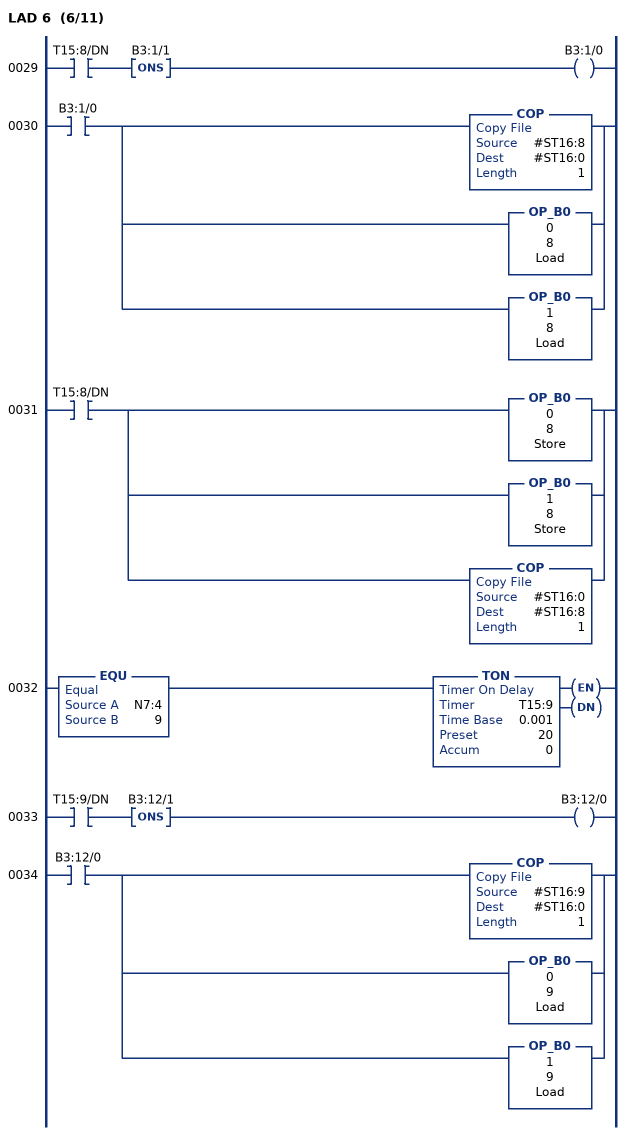
% Rung: 29 %
SOR XIC T15:8/DN ONS B3:1/1 OTE B3:1/0 EOR
% Rung: 30 %
SOR XIC B3:1/0 BST COP #ST16:8 #ST16:0 1 NXB OP_B0 0 8 Load NXB OP_B0 1 8 Load BND EOR
% Rung: 31 %
SOR XIC T15:8/DN BST OP_B0 0 8 Store NXB OP_B0 1 8 Store NXB COP #ST16:0 #ST16:8 1 BND EOR
% Rung: 32 %
SOR EQU N7:4 9 TON T15:9 0.001 20 0 EOR
% Rung: 33 %
SOR XIC T15:9/DN ONS B3:12/1 OTE B3:12/0 EOR
% Rung: 34 %
SOR XIC B3:12/0 BST COP #ST16:9 #ST16:0 1 NXB OP_B0 0 9 Load NXB OP_B0 1 9 Load BND EOR

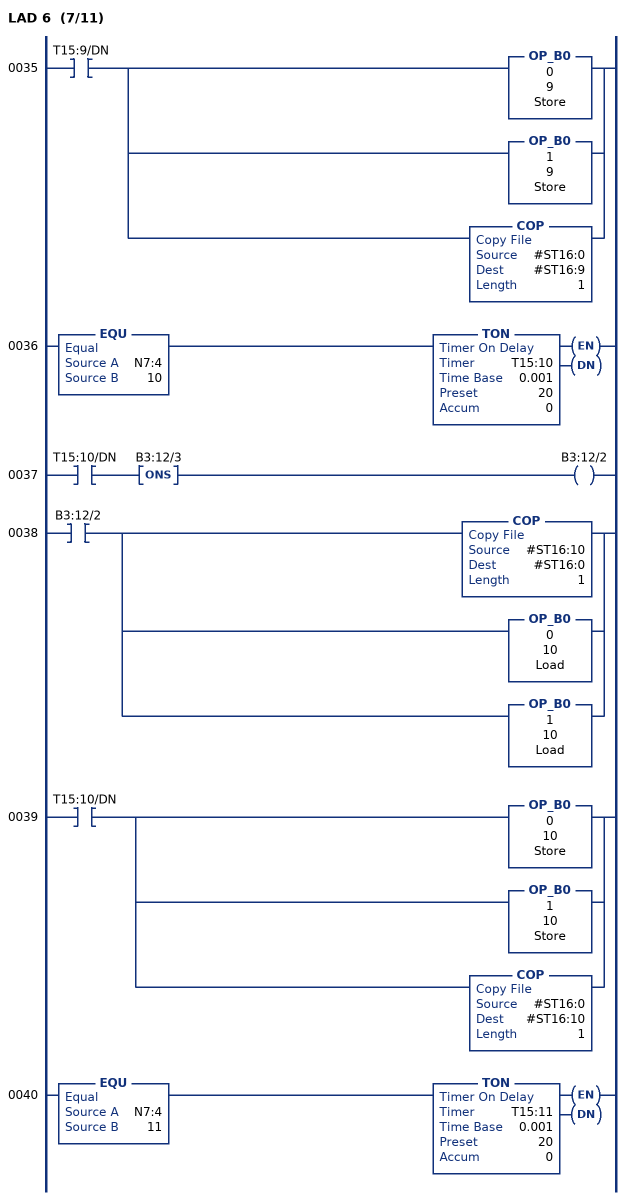
% Rung: 35 %
SOR XIC T15:9/DN BST OP_B0 0 9 Store NXB OP_B0 1 9 Store NXB COP #ST16:0 #ST16:9 1 BND EOR
% Rung: 36 %
SOR EQU N7:4 10 TON T15:10 0.001 20 0 EOR
% Rung: 37 %
SOR XIC T15:10/DN ONS B3:12/3 OTE B3:12/2 EOR
% Rung: 38 %
SOR XIC B3:12/2 BST COP #ST16:10 #ST16:0 1 NXB OP_B0 0 10 Load NXB OP_B0 1 10 Load BND EOR
% Rung: 39 %
SOR XIC T15:10/DN BST OP_B0 0 10 Store NXB OP_B0 1 10 Store NXB COP #ST16:0 #ST16:10 1 BND EOR
% Rung: 40 %
SOR EQU N7:4 11 TON T15:11 0.001 20 0 EOR

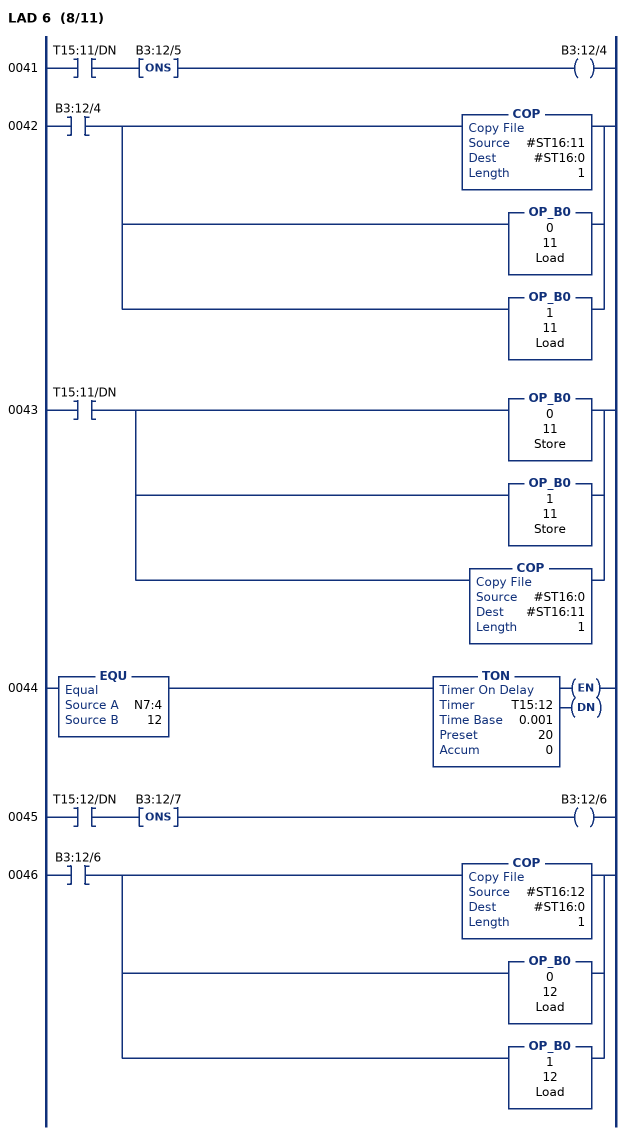
% Rung: 41 %
SOR XIC T15:11/DN ONS B3:12/5 OTE B3:12/4 EOR
% Rung: 42 %
SOR XIC B3:12/4 BST COP #ST16:11 #ST16:0 1 NXB OP_B0 0 11 Load NXB OP_B0 1 11 Load BND EOR
% Rung: 43 %
SOR XIC T15:11/DN BST OP_B0 0 11 Store NXB OP_B0 1 11 Store NXB COP #ST16:0 #ST16:11 1 BND EOR
% Rung: 44 %
SOR EQU N7:4 12 TON T15:12 0.001 20 0 EOR
% Rung: 45 %
SOR XIC T15:12/DN ONS B3:12/7 OTE B3:12/6 EOR
% Rung: 46 %
SOR XIC B3:12/6 BST COP #ST16:12 #ST16:0 1 NXB OP_B0 0 12 Load NXB OP_B0 1 12 Load BND EOR

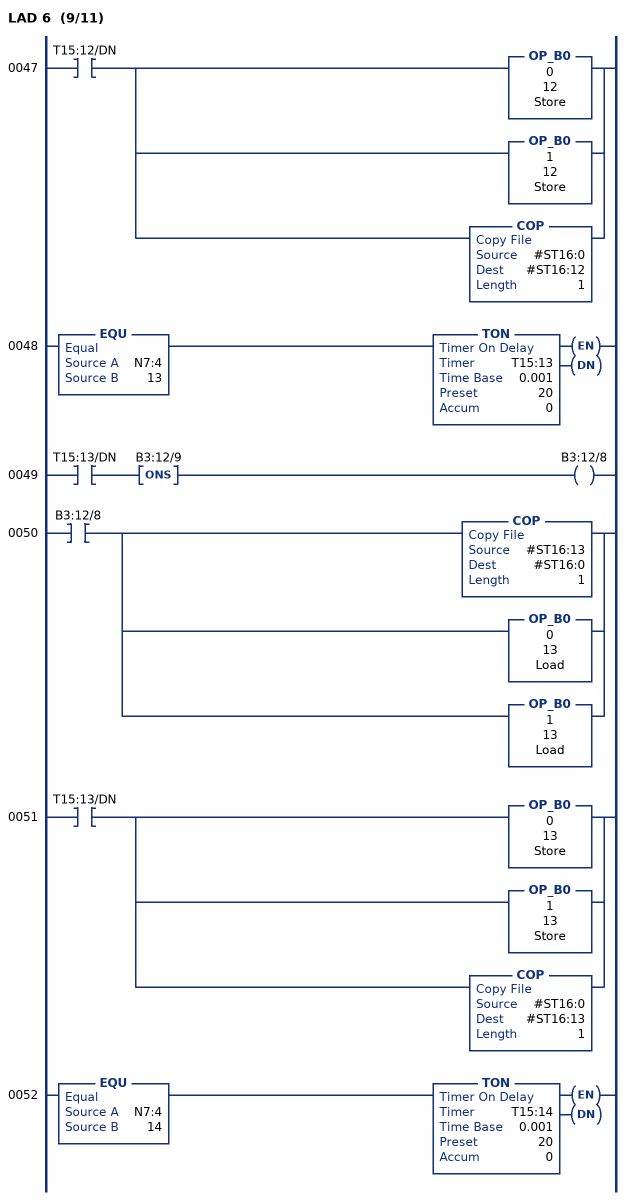
% Rung: 47 %
SOR XIC T15:12/DN BST OP_B0 0 12 Store NXB OP_B0 1 12 Store NXB COP #ST16:0 #ST16:12 1 BND EOR
% Rung: 48 %
SOR EQU N7:4 13 TON T15:13 0.001 20 0 EOR
% Rung: 49 %
SOR XIC T15:13/DN ONS B3:12/9 OTE B3:12/8 EOR
% Rung: 50 %
SOR XIC B3:12/8 BST COP #ST16:13 #ST16:0 1 NXB OP_B0 0 13 Load NXB OP_B0 1 13 Load BND EOR
% Rung: 51 %
SOR XIC T15:13/DN BST OP_B0 0 13 Store NXB OP_B0 1 13 Store NXB COP #ST16:0 #ST16:13 1 BND EOR
% Rung: 52 %
SOR EQU N7:4 14 TON T15:14 0.001 20 0 EOR

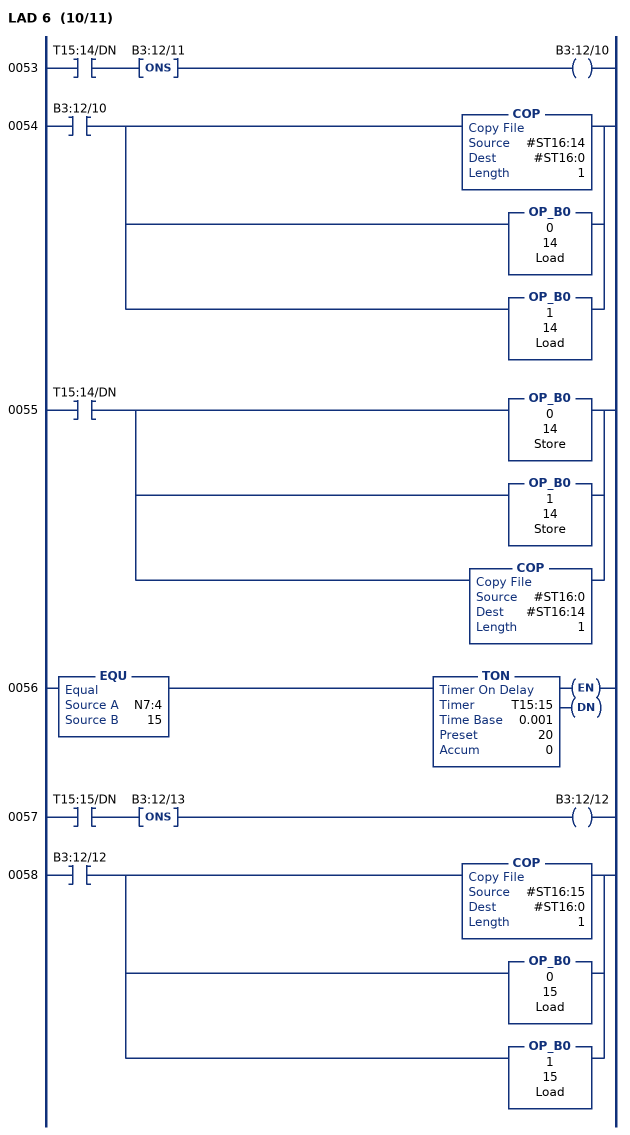
% Rung: 53 %
SOR XIC T15:14/DN ONS B3:12/11 OTE B3:12/10 EOR
% Rung: 54 %
SOR XIC B3:12/10 BST COP #ST16:14 #ST16:0 1 NXB OP_B0 0 14 Load NXB OP_B0 1 14 Load BND EOR
% Rung: 55 %
SOR XIC T15:14/DN BST OP_B0 0 14 Store NXB OP_B0 1 14 Store NXB COP #ST16:0 #ST16:14 1 BND EOR
% Rung: 56 %
SOR EQU N7:4 15 TON T15:15 0.001 20 0 EOR
% Rung: 57 %
SOR XIC T15:15/DN ONS B3:12/13 OTE B3:12/12 EOR
% Rung: 58 %
SOR XIC B3:12/12 BST COP #ST16:15 #ST16:0 1 NXB OP_B0 0 15 Load NXB OP_B0 1 15 Load BND EOR

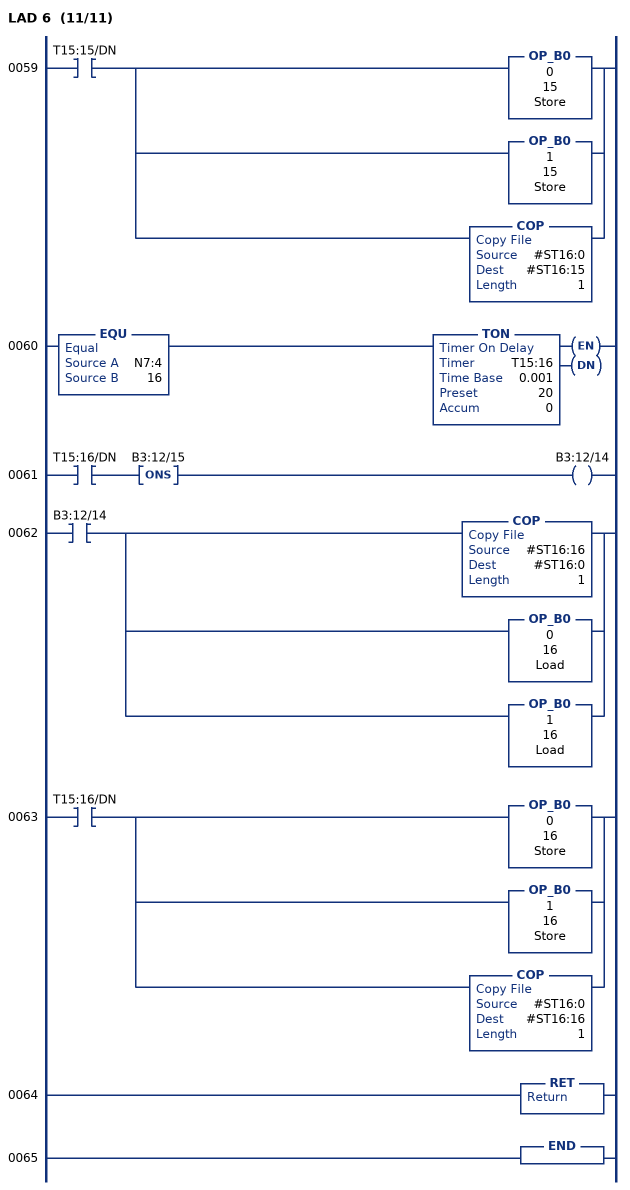
% Rung: 59 %
SOR XIC T15:15/DN BST OP_B0 0 15 Store NXB OP_B0 1 15 Store NXB COP #ST16:0 #ST16:15 1 BND EOR
% Rung: 60 %
SOR EQU N7:4 16 TON T15:16 0.001 20 0 EOR
% Rung: 61 %
SOR XIC T15:16/DN ONS B3:12/15 OTE B3:12/14 EOR
% Rung: 62 %
SOR XIC B3:12/14 BST COP #ST16:16 #ST16:0 1 NXB OP_B0 0 16 Load NXB OP_B0 1 16 Load BND EOR
% Rung: 63 %
SOR XIC T15:16/DN BST OP_B0 0 16 Store NXB OP_B0 1 16 Store NXB COP #ST16:0 #ST16:16 1 BND EOR
% Rung: 64 %
SOR RET EOR
% Rung: 65 %
SOR END EOR

LADDER 18
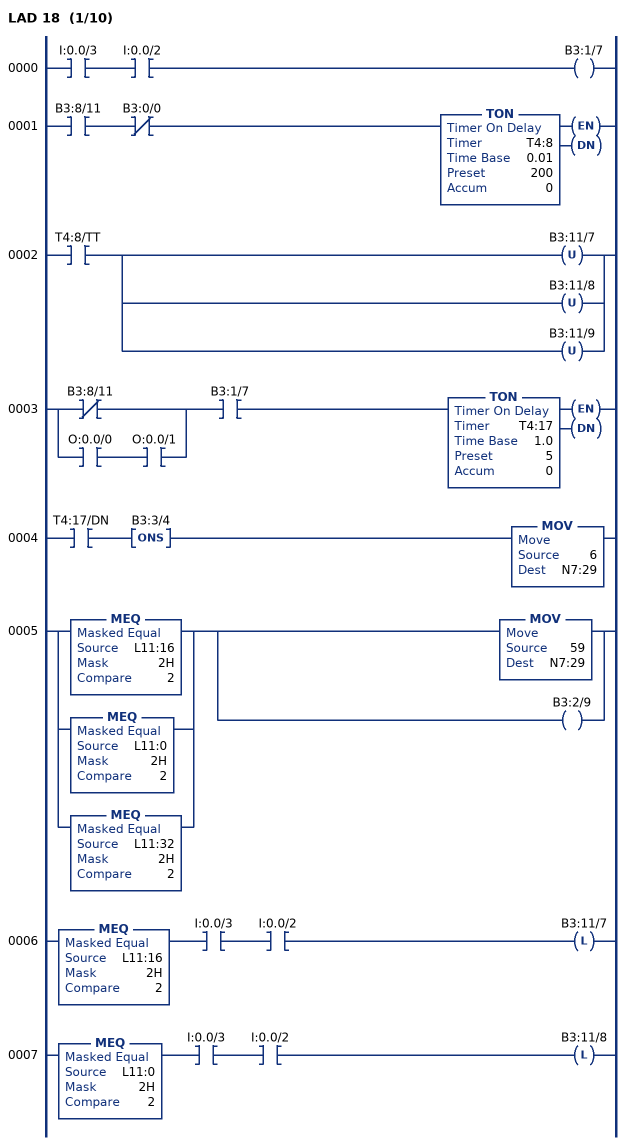
% Rung: 0 %
SOR XIC I:0.0/3 XIC I:0.0/2 OTE B3:1/7 EOR
% Rung: 1 %
SOR XIC B3:8/11 XIO B3:0/0 TON T4:8 0.01 200 0 EOR
% Rung: 2 %
SOR XIC T4:8/TT BST OTU B3:11/7 NXB OTU B3:11/8 NXB OTU B3:11/9 BND EOR
% Rung: 3 %
SOR BST XIO B3:8/11 NXB XIC O:0.0/0 XIC O:0.0/1 BND XIC B3:1/7 TON T4:17 1.0 5 0 EOR
% Rung: 4 %
SOR XIC T4:17/DN ONS B3:3/4 MOV 6 N7:29 EOR
% Rung: 5 %
SOR BST MEQ L11:16 2H 2 NXB MEQ L11:0 2H 2 NXB MEQ L11:32 2H 2 BND BST MOV 59 N7:29 NXB OTE B3:2/9 BND EOR
% Rung: 6 %
SOR MEQ L11:16 2H 2 XIC I:0.0/3 XIC I:0.0/2 OTL B3:11/7 EOR
% Rung: 7 %
SOR MEQ L11:0 2H 2 XIC I:0.0/3 XIC I:0.0/2 OTL B3:11/8 EOR

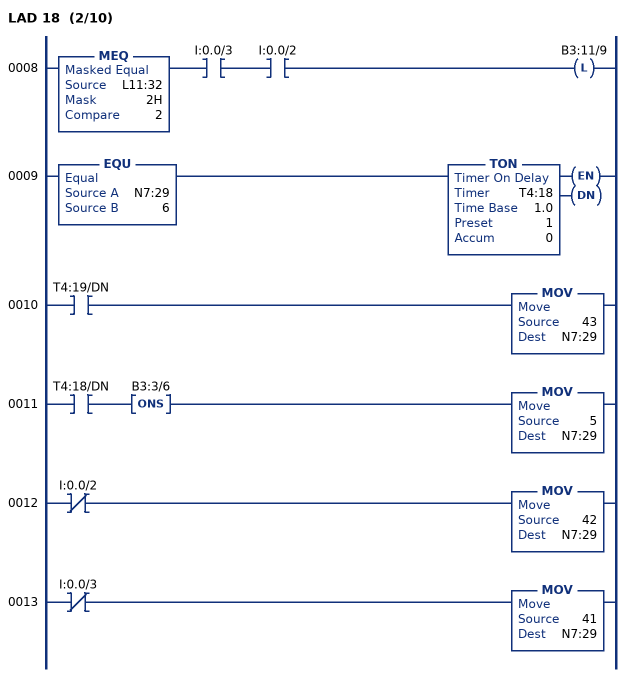
% Rung: 8 %
SOR MEQ L11:32 2H 2 XIC I:0.0/3 XIC I:0.0/2 OTL B3:11/9 EOR
% Rung: 9 %
SOR EQU N7:29 6 TON T4:18 1.0 1 0 EOR
% Rung: 10 %
SOR XIC T4:19/DN MOV 43 N7:29 EOR
% Rung: 11 %
SOR XIC T4:18/DN ONS B3:3/6 MOV 5 N7:29 EOR
% Rung: 12 %
SOR XIO I:0.0/2 MOV 42 N7:29 EOR
% Rung: 13 %
SOR XIO I:0.0/3 MOV 41 N7:29 EOR

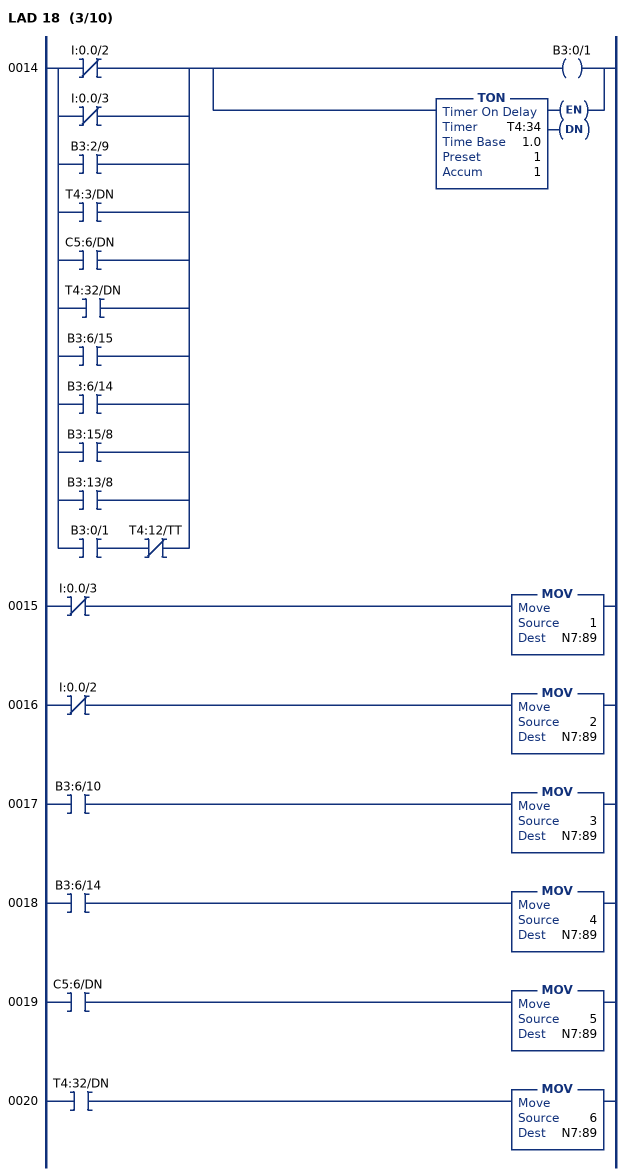
% Rung: 14 %
SOR BST BST XIO I:0.0/2 NXB XIO I:0.0/3 NXB XIC B3:2/9 NXB XIC T4:3/DN NXB XIC C5:6/DN NXB XIC T4:32/DN NXB XIC B3:6/15 NXB XIC B3:6/14 NXB XIC B3:15/8 NXB XIC B3:13/8 BND NXB XIC B3:0/1 XIO T4:12/TT BND BST OTE B3:0/1 NXB TON T4:34 1.0 1 1 BND EOR
% Rung: 15 %
SOR XIO I:0.0/3 MOV 1 N7:89 EOR
% Rung: 16 %
SOR XIO I:0.0/2 MOV 2 N7:89 EOR
% Rung: 17 %
SOR XIC B3:6/10 MOV 3 N7:89 EOR
% Rung: 18 %
SOR XIC B3:6/14 MOV 4 N7:89 EOR
% Rung: 19 %
SOR XIC C5:6/DN MOV 5 N7:89 EOR
% Rung: 20 %
SOR XIC T4:32/DN MOV 6 N7:89 EOR

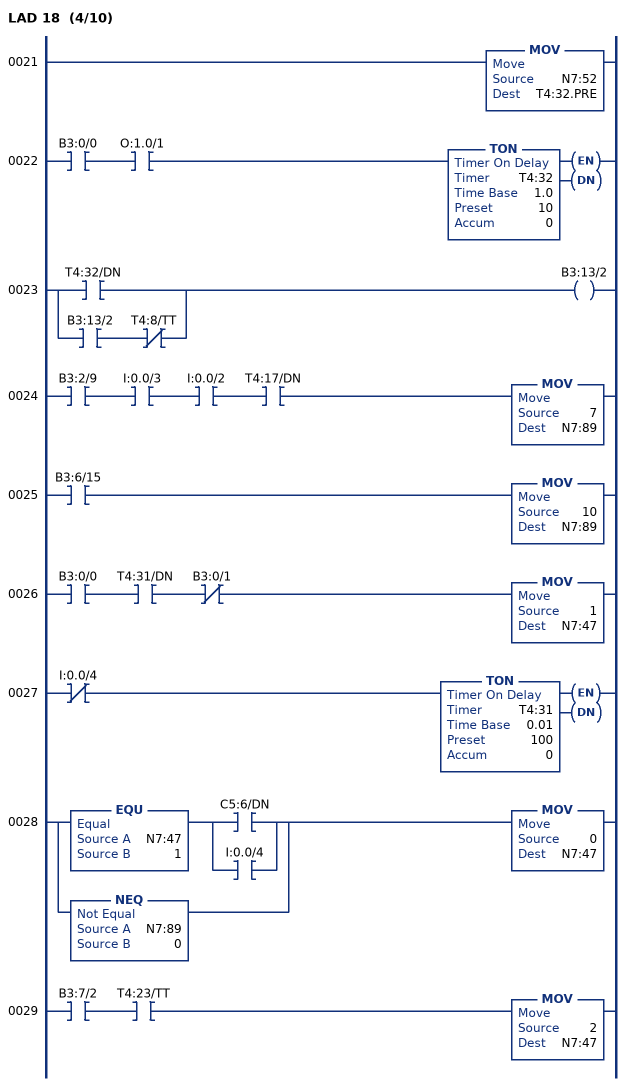
% Rung: 21 %
SOR MOV N7:52 T4:32.PRE EOR
% Rung: 22 %
SOR XIC B3:0/0 XIC O:1.0/1 TON T4:32 1.0 10 0 EOR
% Rung: 23 %
SOR BST XIC T4:32/DN NXB XIC B3:13/2 XIO T4:8/TT BND OTE B3:13/2 EOR
% Rung: 24 %
SOR XIC B3:2/9 XIC I:0.0/3 XIC I:0.0/2 XIC T4:17/DN MOV 7 N7:89 EOR
% Rung: 25 %
SOR XIC B3:6/15 MOV 10 N7:89 EOR
% Rung: 26 %
SOR XIC B3:0/0 XIC T4:31/DN XIO B3:0/1 MOV 1 N7:47 EOR
% Rung: 27 %
SOR XIO I:0.0/4 TON T4:31 0.01 100 0 EOR
% Rung: 28 %
SOR BST EQU N7:47 1 BST XIC C5:6/DN NXB XIC I:0.0/4 BND NXB NEQ N7:89 0 BND MOV 0 N7:47 EOR
% Rung: 29 %
SOR XIC B3:7/2 XIC T4:23/TT MOV 2 N7:47 EOR

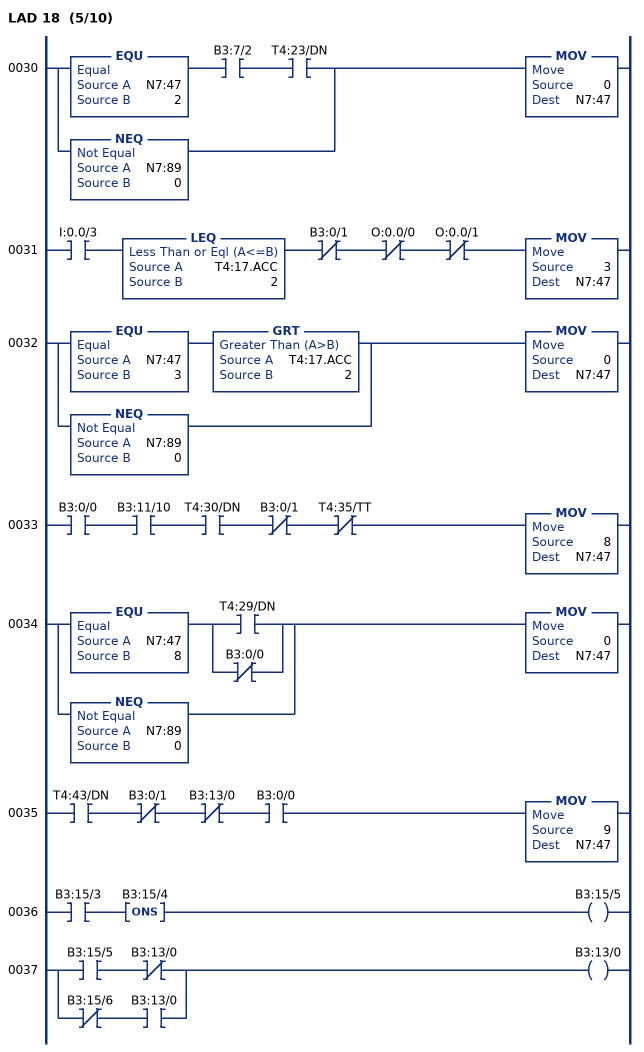
% Rung: 30 %
SOR BST EQU N7:47 2 XIC B3:7/2 XIC T4:23/DN NXB NEQ N7:89 0 BND MOV 0 N7:47 EOR
% Rung: 31 %
SOR XIC I:0.0/3 LEQ T4:17.ACC 2 XIO B3:0/1 XIO O:0.0/0 XIO O:0.0/1 MOV 3 N7:47 EOR
% Rung: 32 %
SOR BST EQU N7:47 3 GRT T4:17.ACC 2 NXB NEQ N7:89 0 BND MOV 0 N7:47 EOR
% Rung: 33 %
SOR XIC B3:0/0 XIC B3:11/10 XIC T4:30/DN XIO B3:0/1 XIO T4:35/TT MOV 8 N7:47 EOR
% Rung: 34 %
SOR BST EQU N7:47 8 BST XIC T4:29/DN NXB XIO B3:0/0 BND NXB NEQ N7:89 0 BND MOV 0 N7:47 EOR
% Rung: 35 %
SOR XIC T4:43/DN XIO B3:0/1 XIO B3:13/0 XIC B3:0/0 MOV 9 N7:47 EOR
% Rung: 36 %
SOR XIC B3:15/3 ONS B3:15/4 OTE B3:15/5 EOR
% Rung: 37 %
SOR BST XIC B3:15/5 XIO B3:13/0 NXB XIO B3:15/6 XIC B3:13/0 BND OTE B3:13/0 EOR

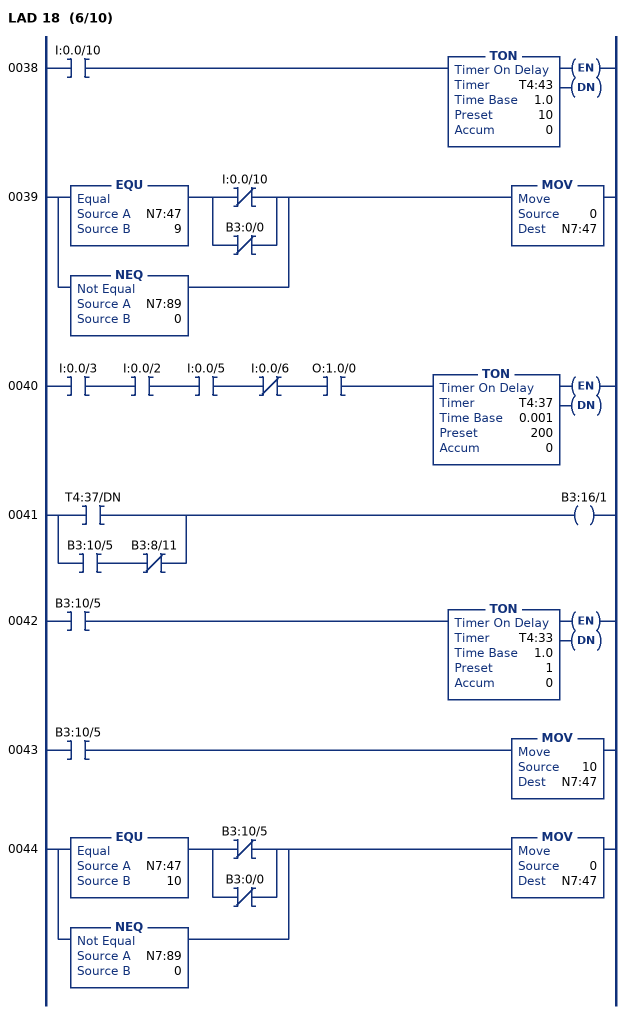
% Rung: 38 %
SOR XIC I:0.0/10 TON T4:43 1.0 10 0 EOR
% Rung: 39 %
SOR BST EQU N7:47 9 BST XIO I:0.0/10 NXB XIO B3:0/0 BND NXB NEQ N7:89 0 BND MOV 0 N7:47 EOR
% Rung: 40 %
SOR XIC I:0.0/3 XIC I:0.0/2 XIC I:0.0/5 XIO I:0.0/6 XIC O:1.0/0 TON T4:37 0.001 200 0 EOR
% Rung: 41 %
SOR BST XIC T4:37/DN NXB XIC B3:10/5 XIO B3:8/11 BND OTE B3:16/1 EOR
% Rung: 42 %
SOR XIC B3:10/5 TON T4:33 1.0 1 0 EOR
% Rung: 43 %
SOR XIC B3:10/5 MOV 10 N7:47 EOR
% Rung: 44 %
SOR BST EQU N7:47 10 BST XIO B3:10/5 NXB XIO B3:0/0 BND NXB NEQ N7:89 0 BND MOV 0 N7:47 EOR

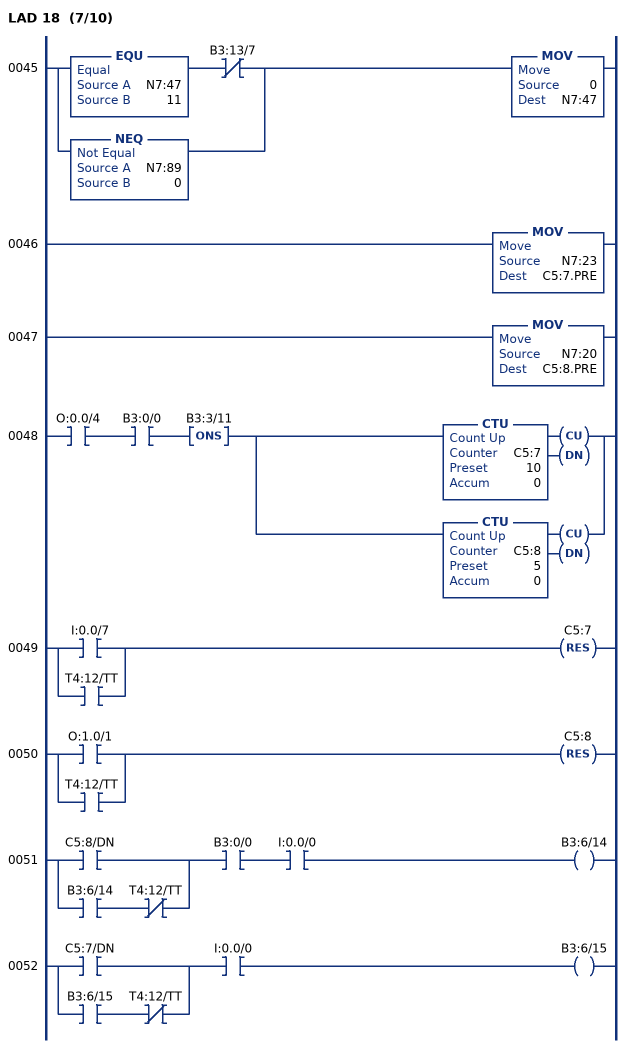
% Rung: 45 %
SOR BST EQU N7:47 11 XIO B3:13/7 NXB NEQ N7:89 0 BND MOV 0 N7:47 EOR
% Rung: 46 %
SOR MOV N7:23 C5:7.PRE EOR
% Rung: 47 %
SOR MOV N7:20 C5:8.PRE EOR
% Rung: 48 %
SOR XIC O:0.0/4 XIC B3:0/0 ONS B3:3/11 BST CTU C5:7 10 0 NXB CTU C5:8 5 0 BND EOR
% Rung: 49 %
SOR BST XIC I:0.0/7 NXB XIC T4:12/TT BND RES C5:7 EOR
% Rung: 50 %
SOR BST XIC O:1.0/1 NXB XIC T4:12/TT BND RES C5:8 EOR
% Rung: 51 %
SOR BST XIC C5:8/DN NXB XIC B3:6/14 XIO T4:12/TT BND XIC B3:0/0 XIC I:0.0/0 OTE B3:6/14 EOR
% Rung: 52 %
SOR BST XIC C5:7/DN NXB XIC B3:6/15 XIO T4:12/TT BND XIC I:0.0/0 OTE B3:6/15 EOR

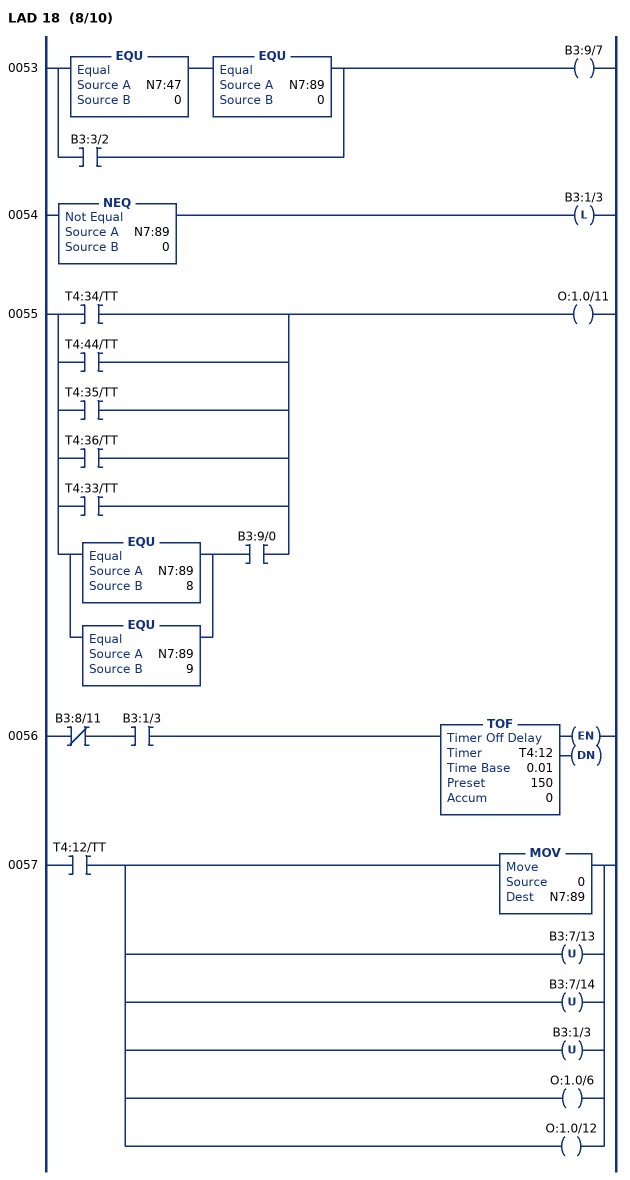
% Rung: 53 %
SOR BST EQU N7:47 0 EQU N7:89 0 NXB XIC B3:3/2 BND OTE B3:9/7 EOR
% Rung: 54 %
SOR NEQ N7:89 0 OTL B3:1/3 EOR
% Rung: 55 %
SOR BST XIC T4:34/TT NXB XIC T4:44/TT NXB XIC T4:35/TT NXB XIC T4:36/TT NXB XIC T4:33/TT NXB BST EQU N7:89 8 NXB EQU N7:89 9 BND XIC B3:9/0 BND OTE O:1.0/11 EOR
% Rung: 56 %
SOR XIO B3:8/11 XIC B3:1/3 TOF T4:12 0.01 150 0 EOR
% Rung: 57 %
SOR XIC T4:12/TT BST MOV 0 N7:89 NXB OTU B3:7/13 NXB OTU B3:7/14 NXB OTU B3:1/3 NXB OTE O:1.0/6 NXB OTE O:1.0/12 BND EOR

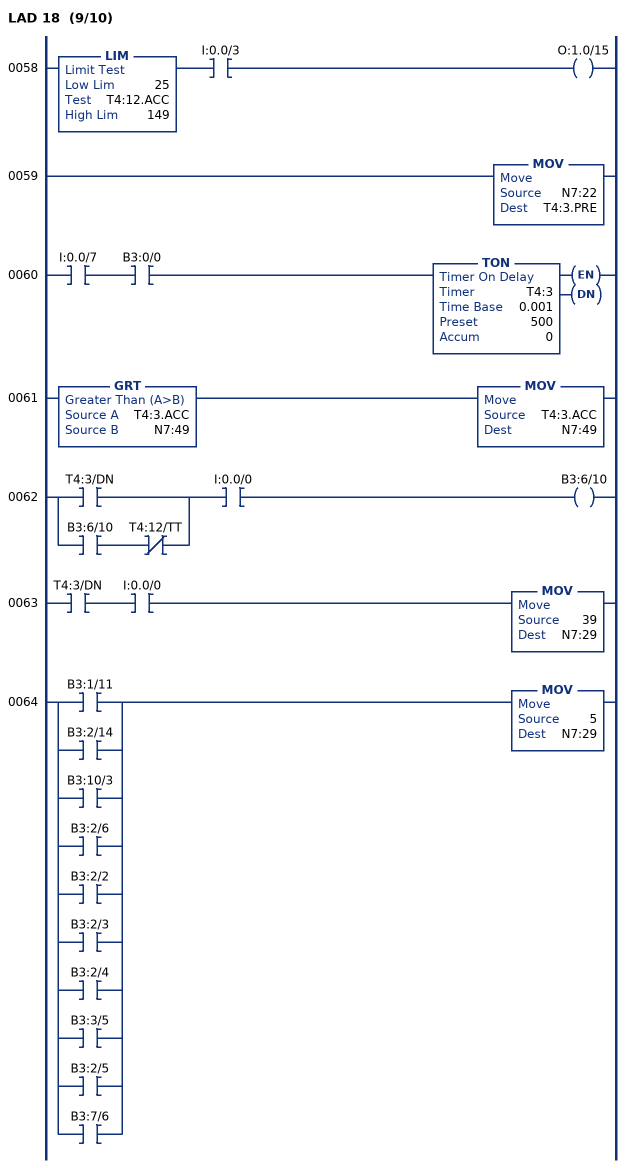
% Rung: 58 %
SOR LIM 25 T4:12.ACC 149 XIC I:0.0/3 OTE O:1.0/15 EOR
% Rung: 59 %
SOR MOV N7:22 T4:3.PRE EOR
% Rung: 60 %
SOR XIC I:0.0/7 XIC B3:0/0 TON T4:3 0.001 500 0 EOR
% Rung: 61 %
SOR GRT T4:3.ACC N7:49 MOV T4:3.ACC N7:49 EOR
% Rung: 62 %
SOR BST XIC T4:3/DN NXB XIC B3:6/10 XIO T4:12/TT BND XIC I:0.0/0 OTE B3:6/10 EOR
% Rung: 63 %
SOR XIC T4:3/DN XIC I:0.0/0 MOV 39 N7:29 EOR
% Rung: 64 %
SOR BST XIC B3:1/11 NXB XIC B3:2/14 NXB XIC B3:10/3 NXB XIC B3:2/6 NXB XIC B3:2/2 NXB XIC B3:2/3 NXB XIC B3:2/4 NXB XIC B3:3/5 NXB XIC B3:2/5 NXB XIC B3:7/6 BND MOV 5 N7:29 EOR

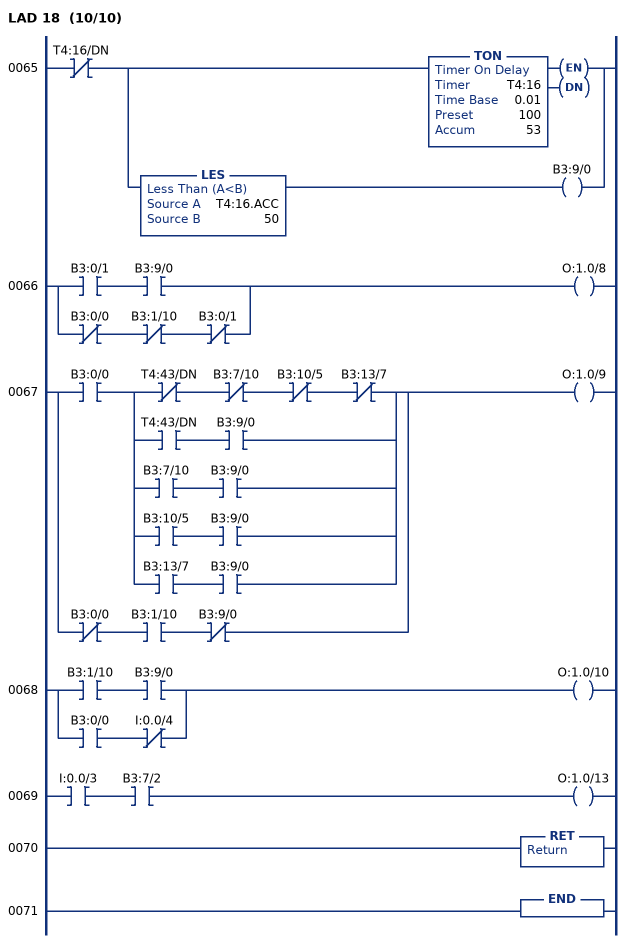
% Rung: 65 %
SOR XIO T4:16/DN BST TON T4:16 0.01 100 53 NXB LES T4:16.ACC 50 OTE B3:9/0 BND EOR
% Rung: 66 %
SOR BST XIC B3:0/1 XIC B3:9/0 NXB XIO B3:0/0 XIO B3:1/10 XIO B3:0/1 BND OTE O:1.0/8 EOR
% Rung: 67 %
SOR BST XIC B3:0/0 BST XIO T4:43/DN XIO B3:7/10 XIO B3:10/5 XIO B3:13/7 NXB XIC T4:43/DN XIC B3:9/0 NXB XIC B3:7/10 XIC B3:9/0 NXB XIC B3:10/5 XIC B3:9/0 NXB XIC B3:13/7 XIC B3:9/0 BND NXB XIO B3:0/0 XIC B3:1/10 XIO B3:9/0 BND OTE O:1.0/9 EOR
% Rung: 68 %
SOR BST XIC B3:1/10 XIC B3:9/0 NXB XIC B3:0/0 XIO I:0.0/4 BND OTE O:1.0/10 EOR
% Rung: 69 %
SOR XIC I:0.0/3 XIC B3:7/2 OTE O:1.0/13 EOR
% Rung: 70 %
SOR RET EOR
% Rung: 71 %
SOR END EOR

DATA TABLE (non-zero values as saved)
DATA B3
% B3:0 % 0X000A 0X0008 0X0400 0X0000 0X0A20 0X0022 0X0008 0X0001 0X0000 0X0E01
% B3:10 % 0X0401 0X007C 0X0000 0X0040 0X0000 0X0000 0X0000 0X0000 0X0000 0X0000
DATA T4
% .PRE .ACC %
% T4:0 % 25 0
% T4:1 % 10000 0
% T4:2 % 5 0
% T4:3 % 500 0
% T4:4 % 50 50
% T4:7 % 50 0
% T4:8 % 200 0
% T4:9 % 1500 0
% T4:10 % 50 0
% T4:11 % 15 0
% T4:12 % 150 0
% T4:13 % 50 0
% T4:14 % 20 21
% T4:15 % 160 0
% T4:16 % 100 53
% T4:17 % 5 0
% T4:18 % 1 0
% T4:19 % 1000 0
% T4:20 % 1 0
% T4:21 % 1 1
% T4:25 % 500 0
% T4:26 % 2 0
% T4:27 % 30 0
% T4:28 % 100 0
% T4:29 % 1000 0
% T4:30 % 100 0
% T4:31 % 100 0
% T4:32 % 10 0
% T4:33 % 1 0
% T4:34 % 1 1
% T4:35 % 1 0
% T4:36 % 1 0
% T4:37 % 200 0
% T4:38 % 2 0
% T4:39 % 5 0
% T4:40 % 50 0
% T4:42 % 30 30
% T4:43 % 10 0
% T4:44 % 1 0
DATA C5
% .PRE .ACC %
% C5:0 % 32000 0
% C5:1 % 32000 0
% C5:2 % 12 0
% C5:3 % 2 0
% C5:4 % 2 0
% C5:5 % 3 0
% C5:6 % 125 0
% C5:7 % 10 0
% C5:8 % 5 0
% C5:9 % 4 0
DATA N7
% N7:0 % 2000 12 0 90 1 160 0 125 100 0
% N7:10 % 34 33 0 1250 250 0 1 125 0 0
% N7:20 % 5 100 500 10 1200 500 400 160 0 41
% N7:30 % 1000 50 50 3 1 50 4970 0 0 250
% N7:40 % 5 3 157 165 157 500 3 0 147 1502
% N7:50 % 1 50 10 1 0 0 0 800 3500 800
% N7:60 % 1000 100 5 10 500 8 1400 1000 5 1700
% N7:70 % 400 0 15 0 140 0 188 40 0 26
% N7:80 % 60 800 1000 400 500 3322 5 10 500 2
% N7:90 % 1000 1000 8 1450 600 0 80 0 173 0
% N7:100 % 188 100 0 10 60 800 3500 800 500 3322
% N7:110 % 75 10 500 10 2000 3000 10 1500 500 0
% N7:120 % 25 0 153 0 66 85 0 26 60 800
% N7:130 % 3500 800 500 3322 100 10 500 15 2000 800
% N7:140 % 5 1500 650 0 35 0 142 0 44 90
% N7:150 % 0 28 60 800 3500 800 500 3322 5 10
% N7:160 % 500 10 1750 1500 800 1750 800 0 15 0
% N7:170 % 129 0 125 56 0 22 60 0 3500 800
% N7:180 % 0 0 100 0 0 10 1500 800 3 1200
% N7:190 % 400 400 30 0 132 0 0 10 0 0
% N7:200 % 0 0 3000 800 0 0 0 207 0 0
% N7:210 % 1500 1000 0 1500 800 0 15 0 123 0
% N7:220 % 0 20 0 0 0 0 3500 800 0 0
% N7:230 % 0 231 0 15 1500 1000 10 1200 500 0
% N7:240 % 15 0 400 50 400 50 400 50 399 70
% N7:250 % 40 84 0 0 0 0
DATA F8
% F8:0 % 0 0 0 0.9235669 250
% F8:5 % 500 500 0.006369427 20.83333 82.83334
% F8:10 % 1.019108 250 4.617835 160 145
% F8:15 % 0 4856.097 3 4855.992 145
% F8:20 % 0.8 1 4855.896 0 4855.997
% F8:25 % 8.333333 50 50 180 2.8
% F8:30 % 100 60 124 35 18
% F8:35 % 76 61 13.00001 13.00001 13.10001
% F8:40 % 12.90001 15 85 60 7
% F8:45 % 1 82 34 64 35
% F8:50 % 60 2.5 20 0 0
% F8:55 % 48 48 0 80 0
% F8:60 % 95 0 0 0
DATA N9
% N9:0 % 34 0 66 22 0 24 60 800 3500 800
% N9:10 % 500 3322 100 10 500 10 2000 1500 3 1500
% N9:20 % 650 0 35 0 37 0 125 18 0 25
% N9:30 % 60 0 2000 800 0 0 100 0 0 20
% N9:40 % 0 1500 5 2000 500 400 15 0 35 0
% N9:50 % 188 67 0 22 60 800 3500 800 500 3322
% N9:60 % 75 10 500 10 2000 3000 10 1400 400 0
% N9:70 % 25 0 110 0 125 30 0 28 60 0
% N9:80 % 3500 800 0 0 100 0 0 10 1500 800
% N9:90 % 3 3500 800 400 30 0
DATA L11
% L11:0 % 844108 -58 -7 0 0
% L11:5 % 0 -1178894336 1167572976 1167572992 0
% L11:10 % 0 -978019930 0 0 0
% L11:15 % 0 844108 -122 -7 0
% L11:20 % 0 0 -1175822336 -987677330 -987677330
% L11:25 % 0 0 -987658416 0 0
% L11:30 % 0 0 842565 -58 -3
% L11:35 % 4 0 0 0 1095761930
% L11:40 % 1095761930 0 1022538569 -1082441984 0
DATA T15
% .PRE .ACC %
% T15:1 % 20 20
% T15:2 % 20 0
% T15:3 % 20 0
% T15:4 % 20 0
% T15:5 % 20 0
% T15:6 % 20 0
% T15:7 % 20 0
% T15:8 % 20 0
% T15:9 % 20 0
% T15:10 % 20 0
% T15:11 % 20 0
% T15:12 % 20 0
% T15:13 % 20 0
% T15:14 % 20 0
% T15:15 % 20 0
% T15:16 % 20 0
% T15:17 % 20 0
% T15:18 % 20 0
% T15:19 % 20 0
% T15:20 % 20 0
% T15:21 % 20 0
% T15:22 % 20 0
% T15:23 % 20 0
% T15:24 % 20 0
% T15:25 % 20 0
% T15:26 % 20 0
% T15:27 % 20 0
% T15:28 % 20 0
% T15:29 % 20 0
% T15:30 % 20 0
% T15:31 % 20 0
% T15:32 % 20 0
% T15:33 % 20 0
% T15:34 % 20 0
% T15:35 % 20 0
% T15:36 % 20 0
% T15:37 % 20 0
% T15:38 % 20 0
% T15:39 % 20 0
% T15:40 % 20 0
DATA ST16
% ST16:2 % "15.2sq oz"
% ST16:3 % "16 oz"
% ST16:4 % "Product 4"
% ST16:5 % "Product 5"
% ST16:6 % "Product 6"
% ST16:7 % "Product 7"
% ST16:8 % "Product 8"
% ST16:9 % "Product 9"
% ST16:10 % "Product 10"
% ST16:11 % "Product 11"
% ST16:12 % "Product 12"
% ST16:13 % "Product 13"
% ST16:14 % "Product 14"
% ST16:15 % "Product 15"
% ST16:16 % "Product 16"
% ST16:17 % "Product 17"
